{attribute 'pack_mode' := '1'}
TYPE ST_1026_Omni_wheels_struct :
STRUCT
	Steer_angle	:REAL;
	Wheel_speed :REAL;
END_STRUCT
END_TYPE

(* stored: Version 1.1.0.1, ProductVersion 3.1.4026.17
   DUT ST_1026_Omni_wheels_struct: Id {c116c078-6ebb-40c4-9433-a8137c6e3714} *)
